ABB RobotStudio station: 210021601057(ziyavudeen).rspag

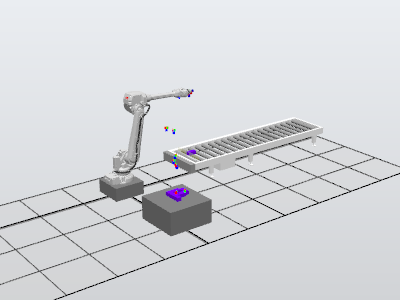
--- station ---
Station Project16 (saved by RobotStudio 23.2.10478.1)
Controller Controller1, task T_ROB1: task frame (RAPID world) sits at (0, 0, 300) mm in the station
Controller Controller1
  mechanical unit ROB_1: IRB4600_40_255_C_01, 6 joints, base frame (0, 0, 0) mm
Layout (positions relative to the parent item):
  - IRB4600_40_255_C_01 [mechanism, from %ABB.RobotStudio.Models.IRB4600%\IRB4600_40_255_C_G_01.rslib] at (0, 0, 300) mm; joint values [0, 0.1705, -0.1152, -3.1416, 0.0579, 3.1416] (rad or m)
  - Conveyor [part, from %ABB.RobotStudio.Models.Conveyors%\Conveyor 950 4000 h2.rslib] at (1600, -425, 0) mm
  - Pedestal [part], size 700 x 700 x 300 mm
  - Attacher [smart component] at (0, -33.08, 1397.68) mm
      signals: DI attach, GO detach
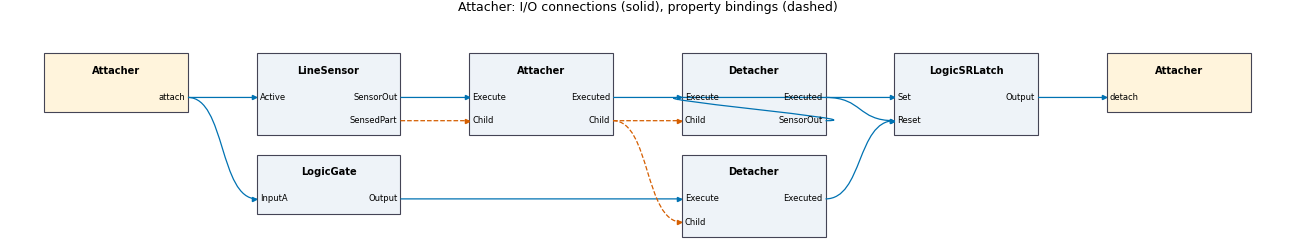
      connections:
        Attacher.attach -> LineSensor.Active
        Attacher.attach -> LogicGate.InputA
        Attacher.Executed -> LogicSRLatch.Set
        Detacher.Executed -> LogicSRLatch.Reset
        LogicSRLatch.Output -> Attacher.detach
        LineSensor.SensorOut -> Attacher.Execute
        PlaneSensor_2.SensorOut -> Detacher.Execute
        LogicGate.Output -> Detacher.Execute
        Detacher.Executed -> LogicSRLatch.Reset
        LineSensor.SensedPart => Attacher.Child
        Attacher.Child => Detacher.Child
        Attacher.Child => Detacher.Child
    - LogicGate [smart component, from Components\LogicGate.rslib]
        properties: Operator=NOT; Delay=0
    - LogicSRLatch [smart component, from Components\LogicSRLatch.rslib]
    - LineSensor [smart component, from Components\LineSensor.rslib] at (1811.16, 51.58, 531.47) mm, rotated rx 180 ry 0.15 rz -180 deg
        properties: Start=[0 0 0]; End=[0 0 0.02]; Length=0.02; Radius=0.0005; Tag=(none); SensedPart=Part_13_86; SensedPoint=[0.28571533203125 -1.67207348632813 0.590785949707031]
      - _sensorPart_ [part], size 1 x 1 x 20 mm
    - Attacher [smart component, from Components\Attacher.rslib]
        properties: Parent=Smart_Gripper_Servo_One_Vacuum; Flange=1; Child=Part_13_86; Mount=false; Offset=[0 0 0]; Orientation=[0 0 0]
    - Smart_Gripper_Servo_One_Vacuum [mechanism, from %ABB.RobotStudio.Models.SmartGripper%\ABB_Smart_Gripper_Servo_One_Vacuum.rslib] at (1773.53, 33.08, 581.37) mm, rotated rx 0 ry 89.85 rz 0 deg; joint values [0] (rad or m)
    - Detacher [smart component, from Components\Detacher.rslib]
        properties: Child=Part_13_86; KeepPosition=true
  - Table [part], size 1000 x 1000 x 500 mm
  - Part_13 [part], size 200 x 100 x 80 mm
  - P [graphiccomponentgroup]
    - Part_6 [part], size 100 x 100 x 80 mm
    - Part_7 [part], size 100 x 100 x 80 mm
    - Part_8 [part], size 100 x 100 x 80 mm
    - Part_9 [part], size 100 x 100 x 80 mm
    - Part_10 [part], size 100 x 100 x 80 mm
    - Part_11 [part], size 100 x 100 x 80 mm
    - Part_12 [part], size 100 x 100 x 80 mm
    - Part_14 [part], size 100 x 200 x 80 mm
  - Conveyor [smart component]
      signals: DO out, DI move
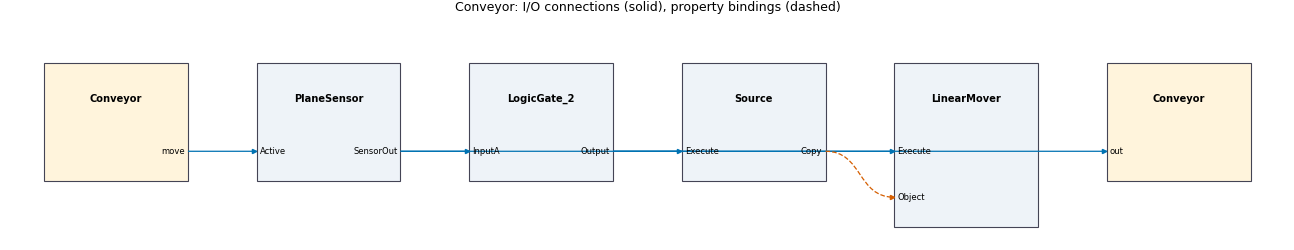
      connections:
        PlaneSensor.SensorOut -> Conveyor.out
        PlaneSensor.SensorOut -> LogicGate_2.InputA
        LogicGate_2.Output -> LinearMover.Execute
        LogicGate_2.Output -> Source.Execute
        Conveyor.move -> PlaneSensor.Active
        Source.Copy => LinearMover.Object
    - PlaneSensor [smart component, from Components\PlaneSensor.rslib]
        properties: Origin=[1.796705 0.43 0.43]; Axis1=[0 0 0.1]; Axis2=[0 -0.8 0]; Tag=(none); SensedPart=Part_13_87
      - _sensorPart_ [part], size 0 x 800 x 100 mm
    - LogicGate_2 [smart component, from Components\LogicGate.rslib]
        properties: Operator=NOT; Delay=0
    - Source [smart component, from Components\Source.rslib]
        properties: Source=Part_13; Copy=Part_13_87; Parent=(none); Position=[0 0 0]; Orientation=[0 0 0]; Transient=false; PhysicsBehavior=-1
    - LinearMover [smart component, from Components\LinearMover.rslib]
        properties: Object=Part_13_87; Direction=[-4 0 0]; Speed=1; Reference=Global; ReferenceObject=(none)
    - SimulationEvents [smart component, from Components\SimulationEvents.rslib]
  - Part_13_82 [part] at (261.08, 3636.95, 62.98) mm, rotated rx -0.96 ry -0.14 rz -89.68 deg, size 200 x 100 x 80 mm
  - Part_13_83 [part] at (-17.63, 3479.62, 74.6) mm, rotated rx 0 ry 0 rz -89.81 deg, size 200 x 100 x 80 mm
  - Part_13_84 [part] at (17.28, 3672.51, -8.86) mm, rotated rx 0.49 ry -0.88 rz -90.14 deg, size 200 x 100 x 80 mm
  - Part_13_85 [part] at (5608.78, -1863.58, 156.3) mm, rotated rx -0.31 ry 0.87 rz 179.3 deg, size 200 x 100 x 80 mm
  - Part_13_86 [part] at (5608.36, -1683.07, 156.5) mm, rotated rx -0.31 ry 0.87 rz 179.3 deg, size 200 x 100 x 80 mm
  - Part_13_87 [part] at (-3504, 0, 0) mm, size 200 x 100 x 80 mm
Attachment: Smart_Gripper_Servo_One_Vacuum is attached to IRB4600_40_255_C_01 / Link6
Attachment: LineSensor is attached to Smart_Gripper_Servo_One_Vacuum / DownFinger
Station logic (signal -> signal, property => property):
  Controller1.di_out -> Attacher.attach
  Conveyor.out -> Controller1.di_inp
  Controller1.di_outt -> Conveyor.move
Targets, tools, work objects and paths stored in the station and not in the controller backup, written as RAPID:
! task T_ROB1
MODULE Module1
  CONST robtarget Target_370:=[[282.526049484,-1560.204987973,984.966004667],[0.00273625,-0.999961716,-0.005493531,-0.006237107],[-1,3,-3,0],[9E+09,9E+09,9E+09,9E+09,9E+09,9E+09]];
  CONST robtarget Target_380:=[[282.525983428,-1560.204862095,984.965886939],[0.002736372,-0.999961715,-0.005493198,-0.006237465],[-1,3,-3,0],[9E+09,9E+09,9E+09,9E+09,9E+09,9E+09]];
  CONST robtarget Target_400:=[[282.52573442,-1850.575262247,293.574117244],[0.002736061,-0.999961716,-0.005493627,-0.00623705],[-1,3,-3,0],[9E+09,9E+09,9E+09,9E+09,9E+09,9E+09]];
  CONST robtarget Target_390:=[[282.525664036,-1850.574986491,318.717569793],[0.002736038,-0.999961716,-0.005493648,-0.006237047],[-1,3,-3,0],[9E+09,9E+09,9E+09,9E+09,9E+09,9E+09]];
ENDMODULE


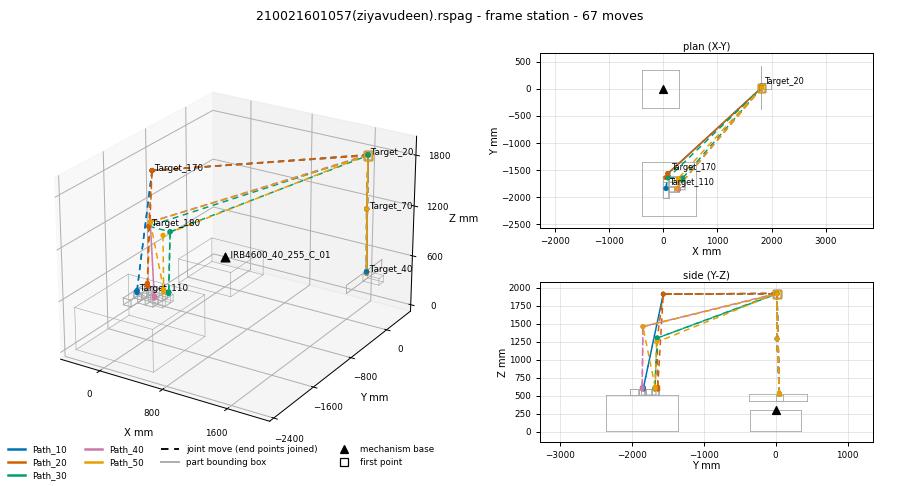
[picture p0: tool path of 210021601057(ziyavudeen).rspag in frame station, 67 of 67 moves have a stored position in this frame; points joined in program order, loops and branches not executed]
--- Controller Data/Controller1/RAPID/TASK1/PROGMOD/CalibData.mod ---
MODULE CalibData
    PERS tooldata Servo:=[TRUE,[[0,0,84],[1,0,0,0]],[0.226,[8.9,12.3,48.7],[1,0,0,0],0.00021,0.00024,0.00009]];
    PERS tooldata VaccumOne:=[TRUE,[[63.5,18.5,37.5],[0.707106781,0,0.707106781,0]],[0.226,[8.9,12.3,48.7],[1,0,0,0],0.00021,0.00024,0.00009]];
ENDMODULE

--- Controller Data/Controller1/RAPID/TASK1/PROGMOD/Module1.mod ---
MODULE Module1
        CONST robtarget Target_10:=[[1562.639382153,18.5,1623.75738686],[0.258819045,0,-0.965925826,0],[-1,-2,1,0],[9E+09,9E+09,9E+09,9E+09,9E+09,9E+09]];
    CONST robtarget Target_20:=[[1811.197060484,18.499998294,1615.643934418],[0.001308987,0.000000003,0.999999143,0],[-1,-2,1,0],[9E+09,9E+09,9E+09,9E+09,9E+09,9E+09]];
    CONST robtarget Target_30:=[[1811.197047271,18.499999254,1615.64344748],[0.001308992,0,0.999999143,0],[0,-2,1,0],[9E+09,9E+09,9E+09,9E+09,9E+09,9E+09]];
    CONST robtarget Target_40:=[[1811.197027919,51.581569383,232.02057786],[0.001308985,0,0.999999143,0],[0,-2,1,0],[9E+09,9E+09,9E+09,9E+09,9E+09,9E+09]];
    CONST robtarget Target_50:=[[1811.197028908,51.58156933,217.967391157],[0.001309014,0,0.999999143,0],[0,-2,1,0],[9E+09,9E+09,9E+09,9E+09,9E+09,9E+09]];
    CONST robtarget Target_60:=[[1811.197027919,51.581569383,232.02057786],[0.001308985,0,0.999999143,0],[0,-2,1,0],[9E+09,9E+09,9E+09,9E+09,9E+09,9E+09]];
    CONST robtarget Target_70:=[[1811.197047271,18.499999254,992.785195727],[0.001308992,0,0.999999143,0],[0,-2,1,0],[9E+09,9E+09,9E+09,9E+09,9E+09,9E+09]];
    CONST robtarget Target_80:=[[1811.197057974,18.499999254,1623.756971562],[0.001309014,0,0.999999143,0],[-1,-3,1,0],[9E+09,9E+09,9E+09,9E+09,9E+09,9E+09]];
    CONST robtarget Target_90:=[[79.584408594,-1809.542305072,1623.756970919],[0.000941094,0.695077889,0.718933248,-0.000909867],[-1,-1,0,1],[9E+09,9E+09,9E+09,9E+09,9E+09,9E+09]];
    CONST robtarget Target_100:=[[43.015169878,-1845.358978492,1018.194977823],[0.000941108,0.695077912,0.718933225,-0.00090988],[-1,-1,0,1],[9E+09,9E+09,9E+09,9E+09,9E+09,9E+09]];
    CONST robtarget Target_110:=[[52.027866017,-1835.369925512,314.330910718],[0.000927178,0.70590251,0.708307795,-0.000924029],[-1,-2,1,0],[9E+09,9E+09,9E+09,9E+09,9E+09,9E+09]];
    CONST robtarget Target_120:=[[52.027866434,-1835.369945463,292.56507673],[0.000927177,0.70590251,0.708307795,-0.000924027],[-1,-2,1,0],[9E+09,9E+09,9E+09,9E+09,9E+09,9E+09]];
    CONST robtarget Target_130:=[[52.027865803,-1835.369914745,314.330811713],[0.000927156,0.70590251,0.708307795,-0.000924008],[-1,-2,1,0],[9E+09,9E+09,9E+09,9E+09,9E+09,9E+09]];
    CONST robtarget Target_140:=[[43.015174211,-1845.358977808,1018.19497763],[0.000941108,0.695077903,0.718933234,-0.00090988],[-1,-1,0,1],[9E+09,9E+09,9E+09,9E+09,9E+09,9E+09]];
    CONST robtarget Target_150:=[[79.584408841,-1809.541957359,1623.756964172],[0.000941091,0.695077905,0.718933232,-0.000909864],[-1,0,-1,1],[9E+09,9E+09,9E+09,9E+09,9E+09,9E+09]];
    CONST robtarget Target_160:=[[1562.639018892,18.499999254,1623.756983853],[0.258819007,0,-0.965925836,0],[-1,-2,1,0],[9E+09,9E+09,9E+09,9E+09,9E+09,9E+09]];
    CONST robtarget Target_170:=[[85.942084121,-1560.20499698,1612.943985095],[0.024409502,-0.723287199,-0.689992701,0.0130337],[-1,-2,1,0],[9E+09,9E+09,9E+09,9E+09,9E+09,9E+09]];
    CONST robtarget Target_180:=[[85.942032583,-1643.015050412,1002.979007578],[0.024409489,-0.723287228,-0.689992671,0.013033681],[-1,0,-1,1],[9E+09,9E+09,9E+09,9E+09,9E+09,9E+09]];
    CONST robtarget Target_190:=[[51.880170872,-1636.472003204,320.949877912],[0.00229183,-0.707945857,-0.706214072,-0.008312428],[-1,0,-1,1],[9E+09,9E+09,9E+09,9E+09,9E+09,9E+09]];
    CONST robtarget Target_200:=[[51.880068038,-1634.168979549,291.346464185],[0.009399719,0.707887159,0.706255041,-0.003351403],[-1,0,-1,1],[9E+09,9E+09,9E+09,9E+09,9E+09,9E+09]];
    CONST robtarget Target_210:=[[51.880170872,-1636.472003204,320.949877912],[0.00229183,-0.707945857,-0.706214072,-0.008312428],[-1,0,-1,1],[9E+09,9E+09,9E+09,9E+09,9E+09,9E+09]];
    CONST robtarget Target_220:=[[360.131678271,-1643.015046091,1002.979001227],[0.02440948,-0.723287204,-0.689992696,0.0130337],[-1,0,-1,1],[9E+09,9E+09,9E+09,9E+09,9E+09,9E+09]];
    CONST robtarget Target_230:=[[353.431834055,-1676.563036654,310.833571464],[0.004170208,-0.70820989,-0.705947563,0.007707112],[-1,0,-1,1],[9E+09,9E+09,9E+09,9E+09,9E+09,9E+09]];
    CONST robtarget Target_240:=[[351.236916355,-1676.563038757,292.823433582],[0.004136164,-0.705087484,-0.709066181,0.007725429],[-1,0,-1,1],[9E+09,9E+09,9E+09,9E+09,9E+09,9E+09]];
    CONST robtarget Target_250:=[[353.431840743,-1676.563004048,310.833545382],[0.004170215,-0.708209862,-0.705947591,0.007707106],[-1,0,-1,1],[9E+09,9E+09,9E+09,9E+09,9E+09,9E+09]];
    CONST robtarget Target_260:=[[85.941968308,-1560.205140786,1612.943994177],[0.007237751,0.006753306,-0.999594243,0.026708739],[-2,2,-4,1],[9E+09,9E+09,9E+09,9E+09,9E+09,9E+09]];
    CONST robtarget Target_270:=[[133.408136891,-1831.135430757,887.532405681],[0.007237614,0.00675321,-0.999594247,0.026708648],[0,-3,1,7],[9E+09,9E+09,9E+09,9E+09,9E+09,9E+09]];
    CONST robtarget Target_280:=[[133.407930248,-1831.134996992,887.532071576],[0.007238139,0.006753537,-0.999594235,0.026708871],[-2,2,-4,1],[9E+09,9E+09,9E+09,9E+09,9E+09,9E+09]];
    CONST robtarget Target_290:=[[116.393352032,-1844.938987531,312.154933346],[0.007606113,-0.007014612,-0.999592414,0.026607297],[0,-4,0,7],[9E+09,9E+09,9E+09,9E+09,9E+09,9E+09]];
    CONST robtarget Target_300:=[[116.393536697,-1844.938941016,292.950165678],[0.007606313,-0.007014272,-0.999592401,0.026607817],[-2,2,-4,1],[9E+09,9E+09,9E+09,9E+09,9E+09,9E+09]];
    CONST robtarget Target_310:=[[116.393354836,-1844.938994523,312.154854243],[0.007606096,-0.007014634,-0.999592415,0.026607244],[0,-4,0,7],[9E+09,9E+09,9E+09,9E+09,9E+09,9E+09]];
    CONST robtarget Target_320:=[[85.941837156,-1560.20490825,1612.944215294],[0.006295285,-0.016541065,-0.999839993,0.002598368],[-2,2,-4,1],[9E+09,9E+09,9E+09,9E+09,9E+09,9E+09]];
    CONST robtarget Target_330:=[[119.327338367,-1828.670031654,912.922296382],[0.006295179,-0.016541061,-0.999839993,0.002598362],[-2,2,-4,1],[9E+09,9E+09,9E+09,9E+09,9E+09,9E+09]];
    CONST robtarget Target_350:=[[119.327121371,-1846.238051891,294.749025596],[0.00629516,-0.016541124,-0.99983999,0.00259924],[-2,2,-4,1],[9E+09,9E+09,9E+09,9E+09,9E+09,9E+09]];
    CONST robtarget Target_340:=[[119.327107323,-1846.23805401,328.047878571],[0.006295249,-0.016541062,-0.999839991,0.002599137],[-2,2,-4,1],[9E+09,9E+09,9E+09,9E+09,9E+09,9E+09]];
    CONST robtarget Target_360:=[[119.326935195,-1846.238195885,328.048030195],[0.006294958,-0.016541495,-0.999839985,0.002599384],[-2,2,-4,1],[9E+09,9E+09,9E+09,9E+09,9E+09,9E+09]];
    CONST robtarget Target_450:=[[286.09076193,-1852.609994106,293.543767642],[0.00266375,-0.999958107,0.00611464,-0.00626899],[-1,-3,3,1],[9E+09,9E+09,9E+09,9E+09,9E+09,9E+09]];
    CONST robtarget Target_430:=[[286.090689214,-1852.609998094,315.965200833],[0.002663764,-0.999958107,0.006114632,-0.006268993],[-1,-3,3,1],[9E+09,9E+09,9E+09,9E+09,9E+09,9E+09]];
    CONST robtarget Target_420:=[[245.467017691,-1842.502006166,1161.754958196],[0.002663657,-0.999958108,0.006114554,-0.006268983],[-1,-1,1,0],[9E+09,9E+09,9E+09,9E+09,9E+09,9E+09]];
    CONST robtarget Target_460:=[[286.090762828,-1852.609993113,315.965135748],[0.002663774,-0.999958107,0.006114626,-0.006268998],[-1,-3,3,1],[9E+09,9E+09,9E+09,9E+09,9E+09,9E+09]];
    CONST robtarget Target_410:=[[85.941753051,-1560.205109277,1612.944008787],[0.002663311,-0.999958111,0.006115317,-0.006267886],[-1,-3,1,0],[9E+09,9E+09,9E+09,9E+09,9E+09,9E+09]];
    CONST robtarget Target_470:=[[275.244510898,-1653.058988073,945.787470632],[0.002663347,-0.999958111,0.006115318,-0.00626791],[-1,-1,1,0],[9E+09,9E+09,9E+09,9E+09,9E+09,9E+09]];
    CONST robtarget Target_480:=[[285.676714854,-1672.088977911,320.661663142],[0.002663201,-0.999958111,0.006115249,-0.006267911],[-1,-1,1,0],[9E+09,9E+09,9E+09,9E+09,9E+09,9E+09]];
    CONST robtarget Target_490:=[[285.676711539,-1672.088974087,293.753144197],[0.002663261,-0.999958111,0.006115244,-0.006267879],[-1,-1,1,0],[9E+09,9E+09,9E+09,9E+09,9E+09,9E+09]];
    CONST robtarget Target_500:=[[285.676714854,-1672.088977911,320.661663142],[0.002663201,-0.999958111,0.006115249,-0.006267911],[-1,-1,1,0],[9E+09,9E+09,9E+09,9E+09,9E+09,9E+09]];
!***********************************************************
    !
    ! Module:  Module1
    !
    ! Description:
    !   <Insert description here>
    !
    ! Author: Mohamed Aadhil T
    !
    ! Version: 1.0
    !
    !***********************************************************


    !***********************************************************
    !
    ! Procedure main
    !
    !   This is the entry point of your program
    !
    !***********************************************************
    PROC main()
        !Add your code here
    ENDPROC
    PROC Path_10()
        MoveJ Target_20,v1000,z100,VaccumOne\WObj:=wobj0;
        MoveJ Target_30,v1000,z100,VaccumOne\WObj:=wobj0;
        MoveJ Target_40,v1000,z100,VaccumOne\WObj:=wobj0;
        MoveJ Target_50,v1000,z100,VaccumOne\WObj:=wobj0;
        WaitTime 2;
        SetDO di_out,1;
        WaitTime 2;
        MoveJ Target_60,v1000,z100,VaccumOne\WObj:=wobj0;
        MoveJ Target_70,v1000,z100,VaccumOne\WObj:=wobj0;
        MoveJ Target_80,v1000,z100,VaccumOne\WObj:=wobj0;
        MoveJ Target_170,v1000,z100,VaccumOne\WObj:=wobj0;
        MoveJ Target_110,v1000,z100,VaccumOne\WObj:=wobj0;
        MoveJ Target_120,v1000,z100,VaccumOne\WObj:=wobj0;
        WaitTime 2;
        SetDO di_out,0;
        SetDO di_outt,1;
        WaitTime 2;
        SetDO di_out,0;
        MoveJ Target_130,v1000,z100,VaccumOne\WObj:=wobj0;
        MoveJ Target_170,v1000,z100,VaccumOne\WObj:=wobj0;
        MoveJ Target_20,v1000,z100,VaccumOne\WObj:=wobj0;
    ENDPROC
    PROC Path_20()
        MoveJ Target_20,v1000,z100,VaccumOne\WObj:=wobj0;
        MoveJ Target_30,v1000,z100,VaccumOne\WObj:=wobj0;
        MoveJ Target_40,v1000,z100,VaccumOne\WObj:=wobj0;
        MoveJ Target_50,v1000,z100,VaccumOne\WObj:=wobj0;
        WaitTime 2;
        SetDO di_out,1;
        WaitTime 2;
        MoveJ Target_60,v1000,z100,VaccumOne\WObj:=wobj0;
        MoveJ Target_70,v1000,z100,VaccumOne\WObj:=wobj0;
        MoveJ Target_80,v1000,z100,VaccumOne\WObj:=wobj0;
        MoveJ Target_170,v1000,z100,VaccumOne\WObj:=wobj0;
        MoveJ Target_180,v1000,z100,VaccumOne\WObj:=wobj0;
        MoveJ Target_190,v1000,z100,VaccumOne\WObj:=wobj0;
        MoveJ Target_200,v1000,z100,VaccumOne\WObj:=wobj0;
        WaitTime 2;
        SetDO di_out,0;
        WaitTime 2;
        MoveJ Target_210,v1000,z100,VaccumOne\WObj:=wobj0;
        MoveJ Target_170,v1000,z100,VaccumOne\WObj:=wobj0;
        MoveJ Target_20,v1000,z100,VaccumOne\WObj:=wobj0;
    ENDPROC
    PROC Path_30()
        MoveJ Target_20,v1000,z100,VaccumOne\WObj:=wobj0;
        MoveJ Target_30,v1000,z100,VaccumOne\WObj:=wobj0;
        MoveJ Target_40,v1000,z100,VaccumOne\WObj:=wobj0;
        MoveJ Target_50,v1000,z100,VaccumOne\WObj:=wobj0;
        WaitTime 2;
        SetDO di_out,1;
        WaitTime 2;
        MoveJ Target_60,v1000,z100,VaccumOne\WObj:=wobj0;
        MoveJ Target_70,v1000,z100,VaccumOne\WObj:=wobj0;
        MoveJ Target_80,v1000,z100,VaccumOne\WObj:=wobj0;
        MoveJ Target_180,v1000,z100,VaccumOne\WObj:=wobj0;
        MoveJ Target_220,v1000,z100,VaccumOne\WObj:=wobj0;
        MoveJ Target_230,v1000,z100,VaccumOne\WObj:=wobj0;
        MoveJ Target_240,v1000,z100,VaccumOne\WObj:=wobj0;
        WaitTime 2;
        SetDO di_out,0;
        WaitTime 2;
        MoveJ Target_250,v1000,z100,VaccumOne\WObj:=wobj0;
        MoveJ Target_220,v1000,z100,VaccumOne\WObj:=wobj0;
        MoveJ Target_20,v1000,z100,VaccumOne\WObj:=wobj0;
    ENDPROC
    PROC Path_40()
        MoveJ Target_20,v1000,z100,VaccumOne\WObj:=wobj0;
        MoveJ Target_30,v1000,z100,VaccumOne\WObj:=wobj0;
        MoveJ Target_40,v1000,z100,VaccumOne\WObj:=wobj0;
        MoveJ Target_50,v1000,z100,VaccumOne\WObj:=wobj0;
        WaitTime 2;
        SetDO di_out,1;
        WaitTime 2;
        MoveJ Target_60,v1000,z100,VaccumOne\WObj:=wobj0;
        MoveJ Target_70,v1000,z100,VaccumOne\WObj:=wobj0;
        MoveJ Target_80,v1000,z100,VaccumOne\WObj:=wobj0;
        MoveJ Target_420,v1000,z100,VaccumOne\WObj:=wobj0;
        MoveJ Target_430,v1000,z100,VaccumOne\WObj:=wobj0;
        MoveJ Target_450,v1000,z100,VaccumOne\WObj:=wobj0;
        WaitTime 2;
        SetDO di_out,0;
        WaitTime 2;
        MoveJ Target_460,v1000,z100,VaccumOne\WObj:=wobj0;
        MoveJ Target_420,v1000,z100,VaccumOne\WObj:=wobj0;
        MoveJ Target_20,v1000,z100,VaccumOne\WObj:=wobj0;
    ENDPROC
    PROC Path_50()
        MoveJ Target_20,v1000,z100,VaccumOne\WObj:=wobj0;
        MoveJ Target_30,v1000,z100,VaccumOne\WObj:=wobj0;
        MoveJ Target_40,v1000,z100,VaccumOne\WObj:=wobj0;
        MoveJ Target_50,v1000,z100,VaccumOne\WObj:=wobj0;
        WaitTime 2;
        SetDO di_out,1;
        WaitTime 2;
        MoveJ Target_60,v1000,z100,VaccumOne\WObj:=wobj0;
        MoveJ Target_70,v1000,z100,VaccumOne\WObj:=wobj0;
        MoveJ Target_80,v1000,z100,VaccumOne\WObj:=wobj0;
        MoveJ Target_470,v1000,z100,VaccumOne\WObj:=wobj0;
        MoveJ Target_480,v1000,z100,VaccumOne\WObj:=wobj0;
        MoveJ Target_490,v1000,z100,VaccumOne\WObj:=wobj0;
        WaitTime 2;
        SetDO di_out,0;
        WaitTime 2;
        MoveJ Target_500,v1000,z100,VaccumOne\WObj:=wobj0;
        MoveJ Target_420,v1000,z100,VaccumOne\WObj:=wobj0;
        MoveJ Target_20,v1000,z100,VaccumOne\WObj:=wobj0;
    ENDPROC
    PROC Final()
        WaitTime 2;
        Path_30;
        Path_10;
        Path_20;
        Path_40;
        Path_50;
    ENDPROC
    PROC Path_60()

    ENDPROC
ENDMODULE

--- Controller Data/Controller1/SYSPAR/EIO.cfg ---
EIO:CFG_1.0:6:1::
#
EIO_SIGNAL:

      -Name "di_inp" -SignalType "DI" -Access "All"

      -Name "di_out" -SignalType "DO" -Access "All"

      -Name "di_outt" -SignalType "DO" -Access "All"
